TYPE
  (* Version 1.0, 2023-03-15, Tim Hesse *)
  ROS2_action_msgs__srv__CancelGoal__Response : STRUCT
    return_code : SINT;
    goals_canceling : ARRAY [0..15] OF ROS2_action_msgs__msg__GoalInfo;
  END_STRUCT;
END_TYPE
